(* CoDeSys 2.3 export: GVL_READ.EXP *)

(* Global variable list: AdsClientTests/GVL_Read *)
VAR_GLOBAL
	StandardTypes 		: ST_StandardTypes;
	StandardArrays 		: ST_StandardArrayTypes;
	ComplexTypes		: ST_ComplexTypes;
	ComplexArrayTypes	: ST_ComplexArrayTypes;
	SpecialTypes		: ST_SpecialTypes;
	IssueSpecificTypes	: ST_IssueSpecificTypes;
END_VAR
